// TIA Portal V18 export
// export: Created 2026-06-08T16:32:20.16844Z, ExportSetting WithDefaults, DisplayName Totally Integrated Automation Portal, DisplayVersion V18, DisplayName TIA Portal Openness, DisplayVersion V18, DisplayName TIA Portal Version Control Interface, DisplayVersion V18, DisplayName STEP 7 Professional, DisplayVersion V18, DisplayName STEP 7 Safety, DisplayVersion V18, DisplayName WinCC Professional, DisplayVersion V18
ORGANIZATION_BLOCK "Main"   // OB1, LAD, ProgramCycle
TITLE = "Main Program Sweep (Cycle)"
VERSION : 0.1
// stored: IsIECCheckEnabled false
   VAR_TEMP
      OB1_EV_CLASS : Byte;   // Bits 0-3 = 1 (Coming event), Bits 4-7 = 1 (Event class 1)
      OB1_SCAN_1 : Byte;   // 1 (Cold restart scan 1 of OB 1), 3 (Scan 2-n of OB 1)
      OB1_PRIORITY : Byte;   // Priority of OB Execution
      OB1_OB_NUMBR : Byte;   // 1 (Organization block 1, OB1)
      OB1_RESERVED_1 : Byte;   // Reserved for system
      OB1_RESERVED_2 : Byte;   // Reserved for system
      OB1_PREV_CYCLE : Int;   // Cycle time of previous OB1 scan (milliseconds)
      OB1_MIN_CYCLE : Int;   // Minimum cycle time of OB1 (milliseconds)
      OB1_MAX_CYCLE : Int;   // Maximum cycle time of OB1 (milliseconds)
      OB1_DATE_TIME : Date_And_Time;   // Date and time OB1 started
   END_VAR
BEGIN

REGION Network 1: LID_PRODUCTION_STATION
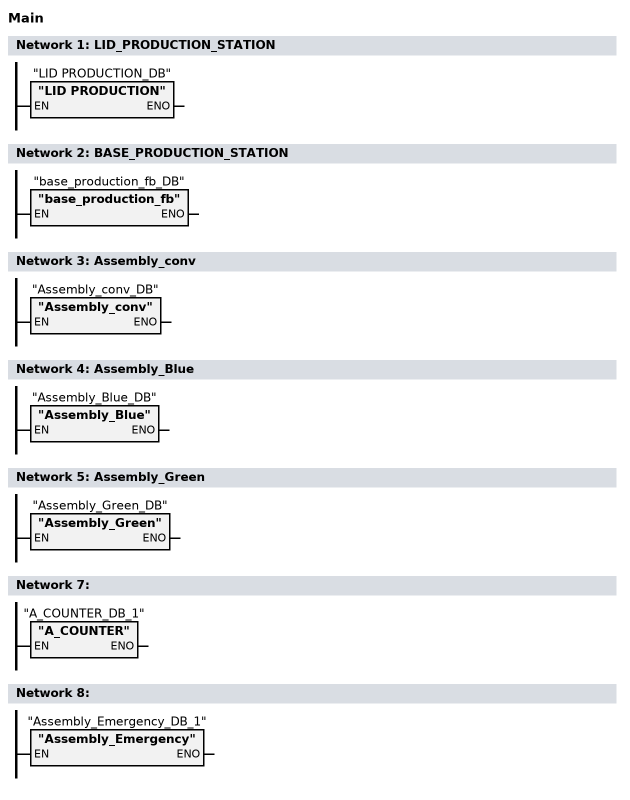
   RUNG wire#powerrail
      "LID PRODUCTION_DB"()
   END_RUNG
   // the same network as SCL:
   "LID PRODUCTION_DB"();   // "LID PRODUCTION"
END_REGION

REGION Network 2: BASE_PRODUCTION_STATION
   RUNG wire#powerrail
      "base_production_fb_DB"()
   END_RUNG
   // the same network as SCL:
   "base_production_fb_DB"();   // "base_production_fb"
END_REGION

REGION Network 3: Assembly_conv
   RUNG wire#powerrail
      "Assembly_conv_DB"()
   END_RUNG
   // the same network as SCL:
   "Assembly_conv_DB"();   // "Assembly_conv"
END_REGION

REGION Network 4: Assembly_Blue
   RUNG wire#powerrail
      "Assembly_Blue_DB"()
   END_RUNG
   // the same network as SCL:
   "Assembly_Blue_DB"();   // "Assembly_Blue"
END_REGION

REGION Network 5: Assembly_Green
   RUNG wire#powerrail
      "Assembly_Green_DB"()
   END_RUNG
   // the same network as SCL:
   "Assembly_Green_DB"();   // "Assembly_Green"
END_REGION

REGION Network 7
   RUNG wire#powerrail
      "A_COUNTER_DB_1"()
   END_RUNG
   // the same network as SCL:
   "A_COUNTER_DB_1"();   // "A_COUNTER"
END_REGION

REGION Network 8
   RUNG wire#powerrail
      "Assembly_Emergency_DB_1"()
   END_RUNG
   // the same network as SCL:
   "Assembly_Emergency_DB_1"();   // "Assembly_Emergency"
END_REGION
END_ORGANIZATION_BLOCK
